# EPICS autosave request: mrfApp/Db/evr-template-dbus-bit-to-pulse-gen.inc.req
$(P)$(R)DBus:B@DBUS_BIT_NUM@:MapTo:TrigPulseGen@PULSE_GEN_NUM@
